% RSLogix 500 project P2_RIZVI_M.RSS, saved by version 8.10.00.18 %
PROJECT "UNTITLED"    % processor: Bul.1763 MicroLogix 1100 Series B %

PROGRAM FILES
  LAD 2 "MAIN"  3 rungs
  LAD 3 "DIGITAL IO"  8 rungs
  LAD 4 "CONTROLS"  5 rungs

DATA FILES
  O0 OUTPUT  4 elements
  I1 INPUT  6 elements
  S2 STATUS  66 elements
  B3 BINARY  1 elements
  T4 TIMER  1 elements
  C5 COUNTER  1 elements
  R6 CONTROL  1 elements
  N7 INTEGER  1 elements
  F8 FLOAT  1 elements

LADDER 2 "MAIN"
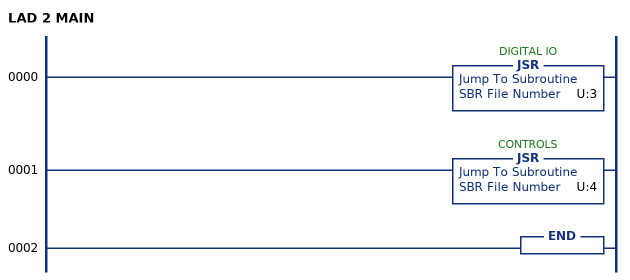
% Rung: 0 %
SOR JSR U:3 EOR
%   U:3  "DIGITAL IO" %
% Rung: 1 %
SOR JSR U:4 EOR
%   U:4  "CONTROLS" %
% Rung: 2 %
SOR END EOR

LADDER 3 "DIGITAL IO"
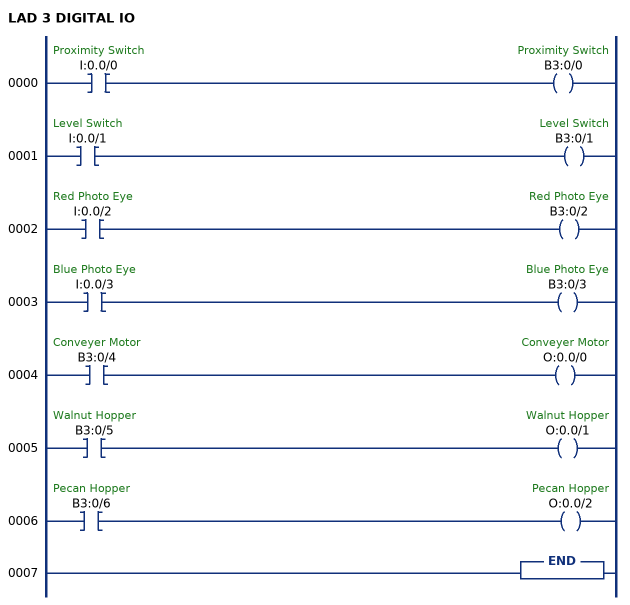
% Rung: 0 %
SOR XIC I:0.0/0 OTE B3:0/0 EOR
%   I:0.0/0  "Proximity Switch" %
%   B3:0/0  "Proximity Switch" %
% Rung: 1 %
SOR XIC I:0.0/1 OTE B3:0/1 EOR
%   I:0.0/1  "Level Switch" %
%   B3:0/1  "Level Switch" %
% Rung: 2 %
SOR XIC I:0.0/2 OTE B3:0/2 EOR
%   I:0.0/2  "Red Photo Eye" %
%   B3:0/2  "Red Photo Eye" %
% Rung: 3 %
SOR XIC I:0.0/3 OTE B3:0/3 EOR
%   I:0.0/3  "Blue Photo Eye" %
%   B3:0/3  "Blue Photo Eye" %
% Rung: 4 %
SOR XIC B3:0/4 OTE O:0.0/0 EOR
%   B3:0/4  "Conveyer Motor" %
%   O:0.0/0  "Conveyer Motor" %
% Rung: 5 %
SOR XIC B3:0/5 OTE O:0.0/1 EOR
%   B3:0/5  "Walnut Hopper" %
%   O:0.0/1  "Walnut Hopper" %
% Rung: 6 %
SOR XIC B3:0/6 OTE O:0.0/2 EOR
%   B3:0/6  "Pecan Hopper" %
%   O:0.0/2  "Pecan Hopper" %
% Rung: 7 %
SOR END EOR

LADDER 4 "CONTROLS"
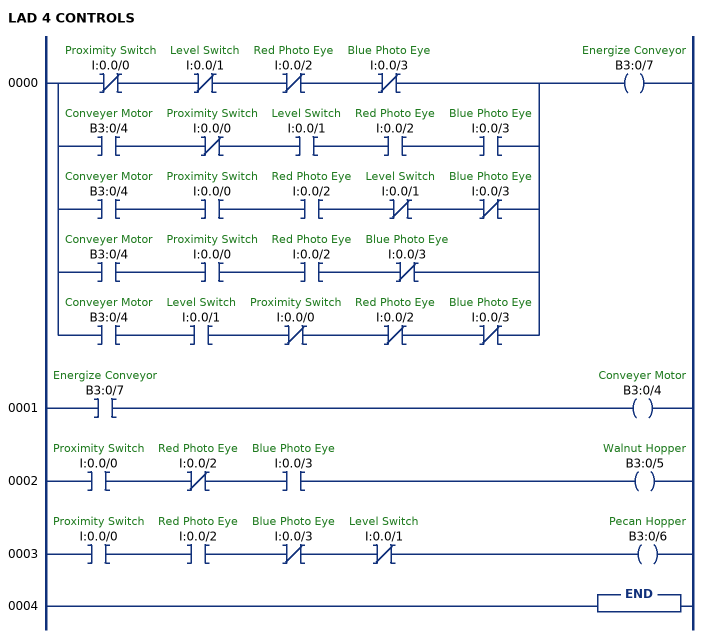
% Rung: 0 %
SOR BST BST BST BST XIO I:0.0/0 XIO I:0.0/1 XIO I:0.0/2 XIO I:0.0/3 NXB XIC B3:0/4 XIO I:0.0/0 XIC I:0.0/1 XIC I:0.0/2 XIC I:0.0/3 BND NXB XIC B3:0/4 XIC I:0.0/0 XIC I:0.0/2 XIO I:0.0/1 XIO I:0.0/3 BND NXB XIC B3:0/4 XIC I:0.0/0 XIC I:0.0/2 XIO I:0.0/3 BND NXB XIC B3:0/4 XIC I:0.0/1 XIO I:0.0/0 XIO I:0.0/2 XIO I:0.0/3 BND OTE B3:0/7 EOR
%   I:0.0/0  "Proximity Switch" %
%   I:0.0/1  "Level Switch" %
%   I:0.0/2  "Red Photo Eye" %
%   I:0.0/3  "Blue Photo Eye" %
%   B3:0/4  "Conveyer Motor" %
%   B3:0/7  "Energize Conveyor" %
% Rung: 1 %
SOR XIC B3:0/7 OTE B3:0/4 EOR
%   B3:0/7  "Energize Conveyor" %
%   B3:0/4  "Conveyer Motor" %
% Rung: 2 %
SOR XIC I:0.0/0 XIO I:0.0/2 XIC I:0.0/3 OTE B3:0/5 EOR
%   I:0.0/0  "Proximity Switch" %
%   I:0.0/2  "Red Photo Eye" %
%   I:0.0/3  "Blue Photo Eye" %
%   B3:0/5  "Walnut Hopper" %
% Rung: 3 %
SOR XIC I:0.0/0 XIC I:0.0/2 XIO I:0.0/3 XIO I:0.0/1 OTE B3:0/6 EOR
%   I:0.0/0  "Proximity Switch" %
%   I:0.0/2  "Red Photo Eye" %
%   I:0.0/3  "Blue Photo Eye" %
%   I:0.0/1  "Level Switch" %
%   B3:0/6  "Pecan Hopper" %
% Rung: 4 %
SOR END EOR
